(* PLC project VisuTest.project, CODESYS CODESYS V3.5 SP17 Patch 2 *)
(* stored: creationDateTime 2022-02-17T09:26:16.669529, modificationDateTime 2022-02-16T16:05:59.7420926 *)

CONFIGURATION 
END_CONFIGURATION
